// TIA Portal project "babu_5LampOnAnd10Off" (V15)

(* hardware
DEVICE "S7-1200 station_1"  S7-1200 Station
   slot 0: "Rack_0"  S7-1200 Rack  Rack  V1.0
   slot 1: "PLC_1"  CPU 1212C DC/DC/DC  6ES7 212-1AE40-0XB0  V4.2
*)

// ===== PLC "PLC_1"  CPU 1212C DC/DC/DC =====

VAR_GLOBAL   // PLC tag table "Default tag table"
   "PUSH BUTTON" AT %M0.0 : Bool;
   "PUSH BUTTON MEMORY" AT %M0.1 : Bool;
   "PULSE" AT %M0.2 : Bool;
   "PULSE ON" AT %M0.3 : Bool;
   "LAMP MEM" AT %M0.4 : Bool;
   "10S MEM" AT %M0.5 : Bool;
   "5S MEM" AT %M0.6 : Bool;
   "RESET COUNTERS" AT %M0.7 : Bool;
   "LAMP" AT %Q0.0 : Bool;
END_VAR

// folder: System blocks/Program resources

DATA_BLOCK "IEC_Timer_0_DB"   // DB1
{ S7_Optimized_Access := 'TRUE' }
AUTHOR : Simatic
FAMILY : IEC
NAME : IEC_TMR
VERSION : 1.0
// stored: InstanceOfName IEC_TIMER
"IEC_TIMER"
BEGIN
END_DATA_BLOCK

DATA_BLOCK "IEC_Timer_0_DB_1"   // DB2
{ S7_Optimized_Access := 'TRUE' }
AUTHOR : Simatic
FAMILY : IEC
NAME : IEC_TMR
VERSION : 1.0
// stored: InstanceOfName IEC_TIMER
"IEC_TIMER"
BEGIN
END_DATA_BLOCK

DATA_BLOCK "IEC_Timer_0_DB_2"   // DB3
{ S7_Optimized_Access := 'TRUE' }
AUTHOR : Simatic
FAMILY : IEC
NAME : IEC_TMR
VERSION : 1.0
// stored: InstanceOfName IEC_TIMER
"IEC_TIMER"
BEGIN
END_DATA_BLOCK

DATA_BLOCK "IEC_Counter_0_DB"   // DB4
{ S7_Optimized_Access := 'TRUE' }
AUTHOR : Simatic
FAMILY : IEC
NAME : CNTR
VERSION : 1.0
// stored: InstanceOfName IEC_COUNTER
"IEC_COUNTER"
BEGIN
END_DATA_BLOCK

DATA_BLOCK "IEC_Counter_0_DB_1"   // DB5
{ S7_Optimized_Access := 'TRUE' }
AUTHOR : Simatic
FAMILY : IEC
NAME : CNTR
VERSION : 1.0
// stored: InstanceOfName IEC_COUNTER
"IEC_COUNTER"
BEGIN
END_DATA_BLOCK

// folder: (top level)

ORGANIZATION_BLOCK "Main"   // OB1, LAD, ProgramCycle
TITLE = "Main Program Sweep (Cycle)"
{ S7_Optimized_Access := 'TRUE' }
VERSION : 0.1
   VAR_INPUT
      Initial_Call : Bool;   // Initial call of this OB
      Remanence : Bool;   // =True, if remanent data are available
   END_VAR
   VAR_TEMP   // added for the SCL form of the ladder/FBD networks
      _w1 : Bool;
   END_VAR
BEGIN

REGION Network 1
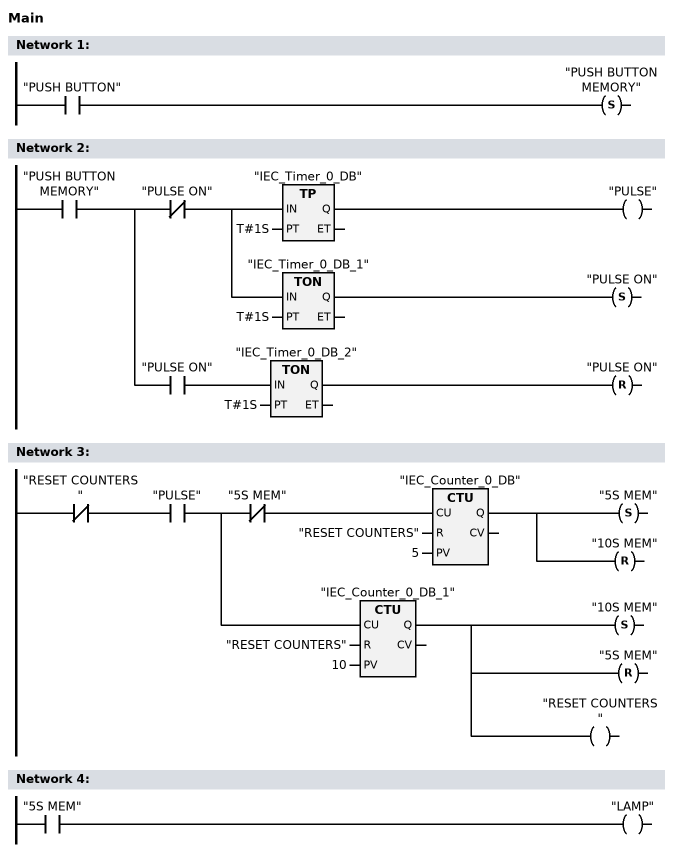
   RUNG wire#powerrail
      Contact( "PUSH BUTTON" )
      S_Coil( "PUSH BUTTON MEMORY" )
   END_RUNG
   // the same network as SCL:
   IF "PUSH BUTTON" THEN "PUSH BUTTON MEMORY" := TRUE; END_IF;
END_REGION

REGION Network 2
   #_w1 := "PUSH BUTTON MEMORY" AND NOT "PULSE ON";
   "IEC_Timer_0_DB".TP(IN := #_w1, PT := T#1S);
   "PULSE" := "IEC_Timer_0_DB".Q;
   "IEC_Timer_0_DB_1".TON(IN := #_w1, PT := T#1S);
   IF "IEC_Timer_0_DB_1".Q THEN "PULSE ON" := TRUE; END_IF;
   "IEC_Timer_0_DB_2".TON(IN := "PUSH BUTTON MEMORY" AND "PULSE ON", PT := T#1S);
   IF "IEC_Timer_0_DB_2".Q THEN "PULSE ON" := FALSE; END_IF;
END_REGION

REGION Network 3
   #_w1 := NOT "RESET COUNTERS" AND "PULSE";
   "IEC_Counter_0_DB".CTU(CU := #_w1 AND NOT "5S MEM", R := "RESET COUNTERS", PV := 5);
   IF "IEC_Counter_0_DB".Q THEN
       "5S MEM" := TRUE;
       "10S MEM" := FALSE;
   END_IF;
   "IEC_Counter_0_DB_1".CTU(CU := #_w1, R := "RESET COUNTERS", PV := 10);
   IF "IEC_Counter_0_DB_1".Q THEN
       "10S MEM" := TRUE;
       "5S MEM" := FALSE;
   END_IF;
   "RESET COUNTERS" := "IEC_Counter_0_DB_1".Q;
END_REGION

REGION Network 4
   RUNG wire#powerrail
      Contact( "5S MEM" )
      Coil( "LAMP" )
   END_RUNG
   // the same network as SCL:
   "LAMP" := "5S MEM";
END_REGION
END_ORGANIZATION_BLOCK